FUNCTION_BLOCK FB_ExampleStation EXTENDS FB_Station
VAR_INPUT
	in_fbDevice : REFERENCE TO FB_Device;
END_VAR
VAR_OUTPUT
END_VAR
VAR
END_VAR

THIS^.A_StateMachine();

END_FUNCTION_BLOCK

(* stored: Version 1.1.0.1, ProductVersion 3.1.4024.11
   POU FB_ExampleStation: Id {77adcf09-04b1-4622-a2a1-1d174c99f352}, SpecialFunc None *)
